Staubli VAL3: robot2PC.pgx

program robot2PC()
begin

  clearBuffer(sktoPC)
  //设置终止符 $
  sioCtrl(sktoPC,"endOfString",36)
  sktoPC="run"

  delay(0.5)
  bIsConnectPC=true
  while true

    if (bIsConnectPC==true)
      sDataPC=sktoPC
    endIf
    delay(0)
  endWhile

end
